// TIA Portal V20 export
DATA_BLOCK "InterfaceSignalsConv_BA40"   // DB329
// stored: InstanceOfName CallInterfaceSignalsConv, InstanceOfType FB
"CallInterfaceSignalsConv"
   // VAR_INPUT
   //    InterfaceTestMode : Bool;
   // END_VAR
   // VAR_OUTPUT
   //    signals_I2S : "typeInspectionToStack";
   //    signals_S2I : "typeStackToInspection";
   // END_VAR
   // VAR_IN_OUT
   //    Comm_I2S : Array[0..95] of Bool;
   //    Comm_S2I : Array[0..95] of Bool;
   //    InterfaceTestButton : "LER_SignalsInput";
   // END_VAR
   // VAR
   //    statWordBuffer_I2S : Array[0..5] of Word;
   //    statWordBuffer_S2I : Array[0..5] of Word;
   // END_VAR
BEGIN
END_DATA_BLOCK
